Fanuc KAREL source: COMPARE_FILE.kl

PROGRAM T
%NOLOCKGROUP
VAR
 v0 : STRING[40]
 v1 : STRING[40]
 v2 : FILE
 v3 : BOOLEAN
 v4 : INTEGER
 v5 : INTEGER
BEGIN
 COMPARE_FILE(v0, v1, v2, v3, v4, v5)
END T
